Yaskawa INFORM job: 000.JBI

/JOB
//NAME 000
//POS
///NPOS 20,20,20,0,0,0
///TOOL 0
///POSTYPE PULSE
///PULSE
C00000=95902,-19559,-65353,-68228,-62443,70439
C00001=95968,1690,-72978,-76829,-57257,78257
C00002=96643,1036,-73382,-77097,-56952,78162
C00003=126959,-22315,-81469,9281,-14857,36875
C00004=130303,-18329,-78578,26111,-18321,29665
C00005=144285,13854,-56584,51164,-49608,19486
C00006=143322,19500,-50026,46258,-52674,19460
C00007=141666,26696,-41180,39278,-57510,19113
C00008=137915,38481,-26581,29273,-65323,18098
C00009=125843,49359,-10142,7641,-72110,8056
C00010=120624,50890,-8050,-372,-73072,3768
C00011=116044,53455,-6965,-6746,-75432,-399
C00012=112222,49666,-11670,-13697,-72791,-335
C00013=104894,36982,-27447,-25965,-64834,-11231
C00014=96159,35527,-38745,-45462,-66466,-16006
C00015=96850,12193,-58759,-53064,-50282,-14223
C00016=105818,804,-59868,-30133,-40705,-20760
C00017=119050,-17910,-74010,11854,-24099,-37431
C00018=135827,-7962,-68903,53184,-44238,-62042
C00019=116865,-4881,-33684,-3254,-73880,-61311
BC00000=878036
BC00001=878036
BC00002=878036
BC00003=878037
BC00004=878037
BC00005=878037
BC00006=878037
BC00007=878037
BC00008=878037
BC00009=878037
BC00010=878036
BC00011=878037
BC00012=878037
BC00013=878037
BC00014=878037
BC00015=878037
BC00016=878037
BC00017=878037
BC00018=878037
BC00019=878037
EC00000=-1746,0
EC00001=-1746,0
EC00002=-1746,0
EC00003=-1743,0
EC00004=-1743,0
EC00005=-1743,0
EC00006=-1743,0
EC00007=-1743,0
EC00008=-1744,0
EC00009=-1744,0
EC00010=-1745,0
EC00011=-1744,0
EC00012=-1744,0
EC00013=-1744,0
EC00014=-1744,0
EC00015=-1744,0
EC00016=-1744,0
EC00017=-1744,0
EC00018=-1744,0
EC00019=-1744,0
//INST
///DATE 2025/05/16 11:47
///ATTR SC,RW
///GROUP1 RB1,BS1
///GROUP2 ST1
NOP
MOVJ C00000 BC00000 VJ=80.00 DEC=20  +MOVJ EC00000 VJ=0.78
MOVJ C00001 BC00001 VJ=80.00 DEC=20  +MOVJ EC00001 VJ=2.00
TIMER T=0.50
MACRO1 MJ#(0) ARGF8
ARCON
WVON WEV#(25)
MOVC C00002 BC00002 V=5.0 DEC=20  +MOVJ EC00002 VJ=80.00
MOVC C00003 BC00003 V=5.0 DEC=20  +MOVJ EC00003 VJ=80.00
MOVC C00004 BC00004 V=5.0 DEC=20  +MOVJ EC00004 VJ=80.00
MOVL C00005 BC00005 V=5.0 DEC=20  +MOVJ EC00005 VJ=80.00
MOVL C00006 BC00006 V=7.5 DEC=20  +MOVJ EC00006 VJ=80.00
MOVL C00007 BC00007 V=6.7 DEC=20  +MOVJ EC00007 VJ=0.78
MOVC C00008 BC00008 V=5.0 DEC=20  +MOVJ EC00008 VJ=80.00
MOVC C00009 BC00009 V=5.0 DEC=20  +MOVJ EC00009 VJ=80.00
WVON WEV#(22)
MOVC C00010 BC00010 V=5.0 DEC=20  +MOVJ EC00010 VJ=80.00
MOVC C00011 BC00011 V=5.0 DEC=20  +MOVJ EC00011 VJ=80.00
WVON WEV#(24)
MOVC C00012 BC00012 V=5.0 DEC=20  +MOVJ EC00012 VJ=80.00
MOVC C00013 BC00013 V=5.0 DEC=20  +MOVJ EC00013 VJ=80.00
MOVL C00014 BC00014 V=5.0 DEC=20  +MOVJ EC00014 VJ=80.00
WVON WEV#(24)
MOVL C00015 BC00015 V=5.8 DEC=20  +MOVJ EC00015 VJ=80.00
MOVC C00016 BC00016 V=5.8 DEC=20  +MOVJ EC00016 VJ=80.00
MOVL C00017 BC00017 V=5.0 DEC=20  +MOVJ EC00017 VJ=80.00
MOVL C00018 BC00018 V=5.0 DEC=20  +MOVJ EC00018 VJ=80.00
ARCOF
WVOF
MOVJ C00019 BC00019 VJ=80.00 DEC=20  +MOVJ EC00019 VJ=80.00
END
